FUNCTION_BLOCK FB_MQTTTelegraf
VAR_INPUT
	(* published message *)
    Topic:			STRING(255) := 'RoboTel';
	Source:			STRING(255) := 'Environment';
	Location:		STRING(255) := 'roof';
	Parameter:		STRING(255);
	Value:			STRING(255);
END_VAR
VAR_OUTPUT
	bPublished:		BOOL := TRUE;
END_VAR
VAR
	//fbMqttClient:	FB_IotMqttClient;
    bSetParameter: 	BOOL := TRUE;
    sPayloadPub: 	STRING(255) := '';
    bConnect:		BOOL := TRUE;
	bSubscribed:	BOOL;
    //fbMessageQueue:	FB_IotMqttMessageQueue;
    //fbMessage      : FB_IotMqttMessage;
END_VAR

 IF bSetParameter THEN
    bSetParameter               := FALSE;
    MQTTCommunication.fbMqttClient.sHostName      := 'primitivo.aip.de';
    MQTTCommunication.fbMqttClient.nHostPort      := 1883;
    MQTTCommunication.fbMqttClient.sClientId      := 'RoboTelPLC'; 
    MQTTCommunication.fbMqttClient.sTopicPrefix   := ''; 
//  fbMqttClient.nKeepAlive     := 60; 
//  fbMqttClient.sUserName      := ;
//  fbMqttClient.sUserPassword  := ; 
//  fbMqttClient.stWill         := ; 
//  fbMqttClient.stTLS          := ;
    MQTTCommunication.fbMqttClient.ipMessageQueue := MQTTCommunication.fbMessageQueue;
END_IF

MQTTCommunication.fbMqttClient.Execute(bConnect);

IF MQTTCommunication.fbMqttClient.bConnected AND bPublished THEN
	sPayloadPub := CONCAT('measurement,host=RoboTel ', Parameter);
	sPayloadPub := CONCAT(sPayloadPub, '=');
	sPayloadPub := CONCAT(sPayloadPub, Value);
	
	bPublished := MQTTCommunication.fbMqttClient.Publish(	
					sTopic:= Topic, 
					pPayload:= ADR(sPayloadPub), 
					nPayloadSize:= LEN2(ADR(sPayloadPub)), // +1 just adds a \x0
					eQoS:= TcIotMqttQos.AtMostOnceDelivery, //TcIotMqttQos.AtMostOnceDelivery,  TcIotMqttQos.ExactlyOnceDelivery
					bRetain:= FALSE, 
					bQueue:= FALSE );
END_IF

END_FUNCTION_BLOCK

(* stored: Version 1.1.0.1, ProductVersion 3.1.4024.9
   POU FB_MQTTTelegraf: Id {bb9cb307-bbdc-4a8e-8a47-c8cb831b125c}, SpecialFunc None *)
